# EPICS autosave request: measComp/measCompApp/Db/measCompWaveformGen_settings.req
$(P)$(R)UserNumPoints
$(P)$(R)IntNumPoints
$(P)$(R)UserDwell
$(P)$(R)IntFrequency
$(P)$(R)ExtTrigger
$(P)$(R)ExtClock
$(P)$(R)Continuous
